TYPE ST_SCANNER_OpState :
STRUCT
	bReady				: BOOL;
	nActiveProgram		: BYTE;
	bAcceptTrigger		: BOOL;
	bCodeChangeActive	: BOOL;
	nActiveTriggers		: INT;
	nExpectedResp			: INT;
	tAcquisitionTime	: TIME;
	nStatusByte			: BYTE;
	nErrorCode			: UDINT;
	nOpState			: BYTE;
END_STRUCT
END_TYPE

(* stored: Version 1.1.0.1, ProductVersion 3.1.4024.15
   DUT ST_SCANNER_OpState: Id {dd19a220-633f-446e-9801-a0512c506713} *)
